(* CoDeSys 2.3 export: FB_FRONTCABINLIGHTS.EXP *)

(* POU new FB:s/FB_frontCabinLights, FBD *)
FUNCTION_BLOCK FB_frontCabinLights
VAR_INPUT
	MOREBRIGHTNESS		:BOOL;
	LESSBRIGHTNESS		:BOOL;
	BRIGHTNESS_STEP		:DINT;
	LIGHTS_ON				:BOOL;
	LIGHTS_OFF				:BOOL;
	MAINSWITCH_ON		:BOOL;
	INIT						:BOOL;
	DOORLOCKED			:BOOL;
	DOORNOTLOCKED		:BOOL;
END_VAR
VAR_OUTPUT
	LIGHTS_ON				:BOOL;
END_VAR
VAR
	fblightCntrl					:FB_cntrlLights;
	fblight2					:FB_cntrlLights;
	ctu1						:CTU;
	rtrig						:R_TRIG;
	pwm						:PWM1000;
	TON						:TON;
END_VAR
VAR_IN_OUT
	LASTBRIGHTNESS		:DINT;
END_VAR
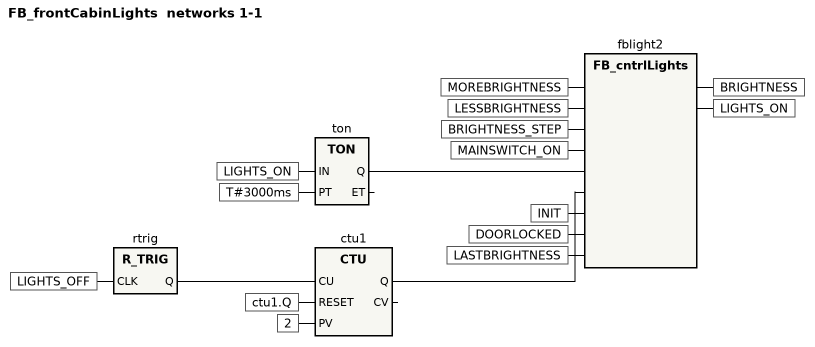
_FBD_ (* Function Block Diagram *)
NETWORK 1
	fblight2:FB_cntrlLights(MOREBRIGHTNESS, LESSBRIGHTNESS, BRIGHTNESS_STEP, MAINSWITCH_ON, ton:TON(IN: LIGHTS_ON, PT: T#3000ms), ctu1:CTU(CU: rtrig:R_TRIG(CLK: LIGHTS_OFF), RESET: ctu1.Q, PV: 2), INIT, DOORLOCKED, LASTBRIGHTNESS, out 2 => LIGHTS_ON) => BRIGHTNESS
_END_FBD_
END_FUNCTION_BLOCK
